{attribute 'qualified_only'}
{attribute 'strict'}
{attribute 'to_string'}
TYPE E_HE_SATT_SequenceState :
(
    IDLE := 0,
    ERROR,
    DETERMINE_FILTER_COMBINATIONS,
    CALCULATE,
    TRIGGER_MOVE_START,
    CONFIRM_MOVE_COMPLETE
);
END_TYPE

(* stored: Version 1.1.0.1
   DUT E_HE_SATT_SequenceState: Id {b241ab8d-0267-4717-89e0-92e9c1826918} *)
